// TwinCAT 3 PLC project PLC
// ProgramVersion: 3.1.4024.0
// libraries:
//   Tc2_MC2, * (Beckhoff Automation GmbH)
//   Tc2_Standard, * (Beckhoff Automation GmbH)
//   Tc2_System, * (Beckhoff Automation GmbH)
//   Tc3_Module, * (Beckhoff Automation GmbH)
// project tree:
//   DUTs/KVM/ ST_KVM.TcDUT, ST_KVM_AC.TcDUT, ST_KVM_App.TcDUT, ST_KVM_CA.TcDUT, ST_KVM_Status.TcDUT
//   GVLs/ GVL.TcGVL, KVM.TcGVL
//   GVLs/IO/ AXIS.TcGVL, INPUT.TcGVL, OUTPUT.TcGVL
//   / PlcTask.TcTTO
//   POUs/ Cartesian.TcPOU, MAIN.TcPOU
//   POUs/KVM/ FB_KVM.TcPOU
// real-time tasks:
//   TASK PlcTask: cycle T#10ms, priority 20, ADS port 350
// motion (NC):
//   TASK NC-Task 1 SAF: cycle T#2ms, priority 4, ADS port 501
//   TASK NC-Task 1 SVB: cycle T#10ms, priority 8, ADS port 511
//   AXIS Axis 1 (id 1)
//     OtherSettings: AllowMotionCmdToSlave=true
//     encoder EncType=1
//     drive DrvType=5
//       Analog: TorqueSetpointScale=10, ScaleFactorActTorque=0.1
//       TimeComp: TaskDelayCycles=1
//     controller CtrType=1
//       CtrPara: PriorControlFactor=1
//         Observer: BandWidth=20
//   AXIS Axis 2 (id 2)
//     OtherSettings: AllowMotionCmdToSlave=true
//     encoder EncType=1
//     drive DrvType=5
//       Analog: TorqueSetpointScale=10, ScaleFactorActTorque=0.1
//       TimeComp: TaskDelayCycles=1
//     controller CtrType=1
//       CtrPara: PriorControlFactor=1
//         Observer: BandWidth=20
//   AXIS Axis 3 (id 3)
//     OtherSettings: AllowMotionCmdToSlave=true
//     encoder EncType=1
//     drive DrvType=5
//       Analog: TorqueSetpointScale=10, ScaleFactorActTorque=0.1
//       TimeComp: TaskDelayCycles=1
//     controller CtrType=1
//       CtrPara: PriorControlFactor=1
//         Observer: BandWidth=20
// variable links:
//   PLC/PLC Instance <-> NC-Task 1 SAF/Axes/Axis 1
//     PlcTask Inputs/AXIS.stAxis1.NcToPlc <-> Outputs/ToPlc
//     PlcTask Outputs/AXIS.stAxis1.PlcToNc <-> Inputs/FromPlc
//   PLC/PLC Instance <-> NC-Task 1 SAF/Axes/Axis 2
//     PlcTask Inputs/AXIS.stAxis2.NcToPlc <-> Outputs/ToPlc
//     PlcTask Outputs/AXIS.stAxis2.PlcToNc <-> Inputs/FromPlc
//   PLC/PLC Instance <-> NC-Task 1 SAF/Axes/Axis 3
//     PlcTask Inputs/AXIS.stAxis3.NcToPlc <-> Outputs/ToPlc
//     PlcTask Outputs/AXIS.stAxis3.PlcToNc <-> Inputs/FromPlc

CONFIGURATION PLC
    RESOURCE PLC ON TwinCAT3
        TASK PlcTask(INTERVAL := T#10ms, PRIORITY := 20);
        PROGRAM MAIN WITH PlcTask : MAIN;
    END_RESOURCE
END_CONFIGURATION

// ---- DUTs/KVM/ST_KVM.TcDUT
TYPE ST_KVM :
STRUCT
	stStatus	: ST_KVM_Status;	// Status
	stApp		: ST_KVM_App;		// Information of application
	stCA		: ST_KVM_CA; 		// Controller -> KVM
	stAC		: ST_KVM_AC;		// KVM -> Controller
END_STRUCT
END_TYPE

// ---- DUTs/KVM/ST_KVM_AC.TcDUT
TYPE ST_KVM_AC :
STRUCT
	boAC			: ARRAY[0..KVM.uiNumOfBool] OF BOOL;
	sboACComments	: ARRAY[0..KVM.uiNumOfBool] OF STRING(20);
	wAC				: ARRAY[0..KVM.uiNumOfWord] OF WORD;
	swACComments	: ARRAY[0..KVM.uiNumOfWord] OF STRING(20);
	lrAC			: ARRAY[0..KVM.uiNumOfDouble] OF LREAL;
	slrACComments	: ARRAY[0..KVM.uiNumOfDouble] OF STRING(20);
END_STRUCT
END_TYPE

// ---- DUTs/KVM/ST_KVM_App.TcDUT
TYPE ST_KVM_App :
STRUCT
	wSID: WORD:=1;	
	wAID: WORD:=1;	
END_STRUCT
END_TYPE

// ---- DUTs/KVM/ST_KVM_CA.TcDUT
TYPE ST_KVM_CA :
STRUCT
	boCA			: ARRAY[0..KVM.uiNumOfBool] OF BOOL;
	sboCAComments	: ARRAY[0..KVM.uiNumOfBool] OF STRING(20);
	wCA				: ARRAY[0..KVM.uiNumOfWord] OF WORD;
	swCAComments	: ARRAY[0..KVM.uiNumOfWord] OF STRING(20);
	lrCA			: ARRAY[0..KVM.uiNumOfDouble] OF LREAL;
	slrCAComments	: ARRAY[0..KVM.uiNumOfDouble] OF STRING(20);
END_STRUCT
END_TYPE

// ---- DUTs/KVM/ST_KVM_Status.TcDUT
TYPE ST_KVM_Status :
STRUCT
	boLive: BOOL;
	boAppLive: BOOL;
	boWebLive: BOOL;
END_STRUCT
END_TYPE

// ---- GVLs/GVL.TcGVL
{attribute 'qualified_only'}
VAR_GLOBAL
END_VAR

// ---- GVLs/IO/AXIS.TcGVL
{attribute 'qualified_only'}
VAR_GLOBAL
	stAxis1 : AXIS_REF;
	stAxis2 : AXIS_REF;
	stAxis3 : AXIS_REF;
END_VAR

// ---- GVLs/IO/INPUT.TcGVL
{attribute 'qualified_only'}
VAR_GLOBAL
	iboEmergencyStopBut	: BOOL; // Emergency button of machine
	iboStartBut			: BOOL; // Start button of machine
	iboStopBut			: BOOL; // Stop button of machine
	iboAlarmResetBut	: BOOL; // Alarm reset button
	iboSystemResetBut	: BOOL; // System reset button for safety 
	iboAutoBut			: BOOL; // Auto / Manuel selection button
	iboManFwdBut		: BOOL; // Manuel forward button for selected axis
	iboManBwdBut		: BOOL; // Manuel backward button for selected axis
END_VAR

// ---- GVLs/IO/OUTPUT.TcGVL
{attribute 'qualified_only'}
VAR_GLOBAL
	qboSTO				: BOOL; // Safe torque off
	qboStartLam			: BOOL; // Lamp of start button
	qboStopLam			: BOOL; // Lamp of stop button
	qboAlarmLam			: BOOL; // Lamp of alarm 
	qboSystemLam		: BOOL; // Lamp of safety
	qboAutoLam			: BOOL; // Lamp of auto button
	qboManFwdLam		: BOOL; // Lamp of forward button
	qboManBwdLam		: BOOL; // Lamp of backward button
END_VAR

// ---- GVLs/KVM.TcGVL
{attribute 'qualified_only'}
VAR_GLOBAL
	gstKVM: ST_KVM;
END_VAR
VAR_GLOBAL CONSTANT
	uiNumOfDouble: INT := 7;
	uiNumOfWord: INT := 7;
	uiNumOfBool: INT := 31;
END_VAR

// ---- POUs/MAIN.TcPOU
PROGRAM MAIN
VAR
	fbKVM: FB_KVM;
	fbCartesian: Cartesian;
END_VAR

fbKVM(wAID:=1 );

fbCartesian(
	boEnable:=INPUT.iboEmergencyStopBut , 
	boStartAck=> , 	
	boEnabAck=> );

END_PROGRAM

// ---- POUs/KVM/FB_KVM.TcPOU
FUNCTION_BLOCK FB_KVM
VAR_INPUT
	wAID: WORD;
END_VAR
VAR_OUTPUT
END_VAR
VAR
	fbTonLive: TON;
	ftriboSystemResetBut: F_TRIG;
END_VAR

IF fbTonLive.Q THEN	KVM.gstKVM.stStatus.boLive:=NOT KVM.gstKVM.stStatus.boLive; END_IF
fbTonLive(IN:=NOT fbTonLive.Q , PT:=T#500MS , Q=> , ET=> );

// AID - Application ID
KVM.gstKVM.stApp.wAID:=wAID;

// selection of application
IF 		wAID=1 THEN	App1();
ELSIF 	wAID=2 THEN	App2(); END_IF

Safety();
General();

ACTION App1:
;
END_ACTION

ACTION App2:
;
END_ACTION

ACTION General:

KVM.gstKVM.stCA.lrCA[0]:=Axis.stAxis1.NcToPlc.ActPos;

INPUT.iboEmergencyStopBut:=KVM.gstKVM.stAC.boAC[0];
INPUT.iboStartBut:=KVM.gstKVM.stAC.boAC[1];
INPUT.iboStopBut:=KVM.gstKVM.stAC.boAC[2];
INPUT.iboAlarmResetBut:=KVM.gstKVM.stAC.boAC[3];
INPUT.iboSystemResetBut:=KVM.gstKVM.stAC.boAC[4];
INPUT.iboAutoBut:=KVM.gstKVM.stAC.boAC[5];
INPUT.iboManFwdBut:=KVM.gstKVM.stAC.boAC[6];
INPUT.iboManBwdBut:=KVM.gstKVM.stAC.boAC[7];

KVM.gstKVM.stCA.boCA[0]:=OUTPUT.qboSTO;
KVM.gstKVM.stCA.boCA[1]:=OUTPUT.qboStartLam;
KVM.gstKVM.stCA.boCA[2]:=OUTPUT.qboStopLam;
KVM.gstKVM.stCA.boCA[3]:=OUTPUT.qboAlarmLam;
KVM.gstKVM.stCA.boCA[4]:=OUTPUT.qboSystemLam;
KVM.gstKVM.stCA.boCA[5]:=OUTPUT.qboAutoLam;
KVM.gstKVM.stCA.boCA[6]:=OUTPUT.qboManFwdLam;
KVM.gstKVM.stCA.boCA[7]:=OUTPUT.qboManBwdLam;
END_ACTION

ACTION Safety:
ftriboSystemResetBut(CLK:=INPUT.iboSystemResetBut, Q=>);
IF INPUT.iboEmergencyStopBut AND ftriboSystemResetBut.Q THEN
	OUTPUT.qboSTO:=TRUE;
END_IF

IF NOT INPUT.iboEmergencyStopBut THEN
	OUTPUT.qboSTO:=FALSE;
END_IF

OUTPUT.qboSystemLam:=OUTPUT.qboSTO;
END_ACTION

END_FUNCTION_BLOCK

// ---- POUs/Cartesian.TcPOU
FUNCTION_BLOCK Cartesian
VAR_INPUT
	boEnable: BOOL;
END_VAR
VAR_OUTPUT
	boStartAck: BOOL;
	boEnabAck: BOOL;
END_VAR
VAR
	rtrboStart: R_TRIG;
	iState: INT;
	fbMoveAbsolute: MC_MoveAbsolute;
	fbMcPower: MC_Power;
	fbTonGec: TON;
	ftrboEnable: F_TRIG;
END_VAR


rtrboStart(CLK:=INPUT.iboStartBut, Q=>);
IF rtrboStart.Q THEN
	boStartAck:=NOT boStartAck;
END_IF

CASE iState OF
0:
	IF boEnable THEN
		iState:=10;
	END_IF
	
10:
	boEnabAck:=TRUE;
	iState:=100;
	
100:
	IF AXIS.stAxis1.Status.StandStill AND boStartAck THEN
		iState:=1000;
	END_IF
	
1000:
	fbMoveAbsolute.Position:=700;
	fbMoveAbsolute.Execute:=TRUE;
	IF fbMoveAbsolute.Done THEN
		fbMoveAbsolute.Execute:=FALSE;
		iState:=1010;
	END_IF
	
1010:
	fbTonGec.IN:=TRUE;
	IF fbTonGec.Q THEN
		fbTonGec.IN:=FALSE;
		iState:=1020;
	END_IF
	
1020:
	fbMoveAbsolute.Position:=0;
	fbMoveAbsolute.Execute:=TRUE;
	IF fbMoveAbsolute.Done THEN
		fbMoveAbsolute.Execute:=FALSE;
		iState:=1030;
	END_IF
	
1030:
	fbTonGec.IN:=TRUE;
	IF fbTonGec.Q THEN
		fbTonGec.IN:=FALSE;
		iState:=100;
	END_IF
	
END_CASE
ftrboEnable(CLK:=boEnable, Q=>);
IF ftrboEnable.Q THEN
	iState:=0;
	boEnabAck:=FALSE;
	boStartAck:=FALSE;
	fbTonGec.IN:=FALSE;
	fbMoveAbsolute.Execute:=FALSE;
END_IF



Axis.stAxis1.ReadStatus();

fbTonGec(IN:= , PT:=T#1S , Q=> , ET=> );

fbMcPower(
	Axis:=Axis.stAxis1 , 
	Enable:=TRUE , 
	Enable_Positive:=TRUE , 
	Enable_Negative:=TRUE , 
	Override:= , 
	BufferMode:= , 
	Options:= , 
	Status=> , 
	Busy=> , 
	Active=> , 
	Error=> , 
	ErrorID=> );
	
fbMoveAbsolute(
	Axis:=Axis.stAxis1 , 
	Execute:= , 
	Position:= , 
	Velocity:=1500 , 
	Acceleration:=10000 , 
	Deceleration:=10000 , 
	Jerk:=100000 , 
	BufferMode:= , 
	Options:= , 
	Done=> , 
	Busy=> , 
	Active=> , 
	CommandAborted=> , 
	Error=> , 
	ErrorID=> );

END_FUNCTION_BLOCK
